TYPE TestStructure :
STRUCT
	num : INT;
	str : STRING(80);
	arr : ARRAY[0..3] OF REAL;
END_STRUCT
END_TYPE

(* stored: Version 1.1.0.1, ProductVersion 3.1.4024.11
   DUT TestStructure: Id {7aec9f90-3ec0-4b9e-8aa6-dc8b93fe5a2c} *)
